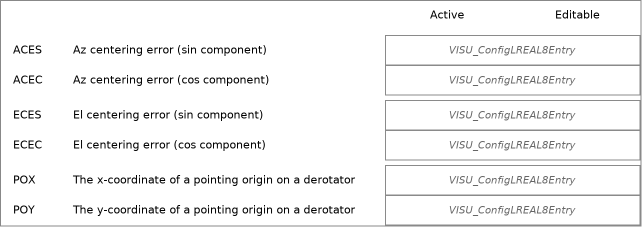
VISUALIZATION VISU_AxesPointingModelConfig_part2  // 642x227
VAR_IN_OUT
    active : AxesPointingModelConfig;
    editable : AxesPointingModelConfig;
END_VAR
    Label (385,5 125x20), "Active"
    Label (515,5 125x20), "Editable"
    Label (10,35 50x30), "ACES"
    Frame (385,35 255x30)
        shows VISU_ConfigLREAL8Entry(active := active.ACES, editable := editable.ACES)
    Label (70,35 315x30), "Az centering error (sin component)"
    Label (10,65 50x30), "ACEC"
    Frame (385,65 255x30)
        shows VISU_ConfigLREAL8Entry(active := active.ACEC, editable := editable.ACEC)
    Label (70,65 315x30), "Az centering error (cos component)"
    Label (10,100 50x30), "ECES"
    Frame (385,100 255x30)
        shows VISU_ConfigLREAL8Entry(active := active.ECES, editable := editable.ECES)
    Label (70,100 315x30), "El centering error (sin component)"
    Label (10,130 50x30), "ECEC"
    Frame (385,130 255x30)
        shows VISU_ConfigLREAL8Entry(active := active.ECEC, editable := editable.ECEC)
    Label (70,130 315x30), "El centering error (cos component)"
    Label (10,165 50x30), "POX"
    Frame (385,165 255x30)
        shows VISU_ConfigLREAL8Entry(active := active.POX, editable := editable.POX)
    Label (70,165 315x30), "The x-coordinate of a pointing origin on a derotator"
    Label (10,195 50x30), "POY"
    Frame (385,195 255x30)
        shows VISU_ConfigLREAL8Entry(active := active.POY, editable := editable.POY)
    Label (70,195 315x30), "The y-coordinate of a pointing origin on a derotator"
END_VISUALIZATION

(* stored: Version 1.1.0.1, ProductVersion 3.1.4019.2
   Visu VISU_AxesPointingModelConfig_part2: Id {b79000d5-2154-40a7-9782-9d4ecdc85b16} *)
